(* Logix 5000 project; controller Wago_EtherNetIP_Adapter_Codesys35 vendor 1 type 14 code 196 rev 32.14; software revision 32.03 *)

TASK MainTask (continuous, watchdog 500 ms) : MainProgram

MODULES
   Local : vendor 1 type 14 code 196 (5069 0, rev 32.14)
      PFC200 : vendor 1285 type 12 code 120 (Ethernet 192.168.2.21, rev 1.1, StandardDataDriven RPI 20 ms)
END_MODULES

VAR_GLOBAL   (* controller tags *)
   AB_to_WAGO_DWORD : DINT := 100;   // DWORD DATA to WAGO PLC
   AB_to_WAGO_REAL : REAL := 7.2;   // REAL DATA to WAGO PLC
   WAGO_to_AB_DWORD : DINT := 500;   // DWORD Data From WAGO PLC
   WAGO_to_AB_REAL : REAL := 1000.0;   // REAL DATA from WAGO PLC
END_VAR

PROGRAM MainProgram   (* main routine MainRoutine *)

ROUTINE MainRoutine   (* ladder *)
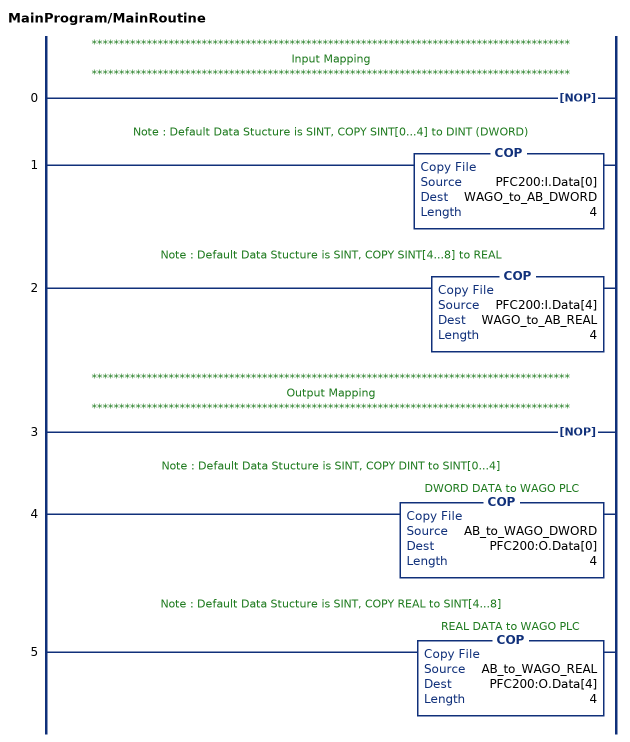
   // ***************************************************************************************
   // Input Mapping
   // ***************************************************************************************
   0: NOP();
   // Note : Default Data Stucture is SINT, COPY SINT[0...4] to DINT (DWORD)
   1: COP(PFC200:I.Data[0],WAGO_to_AB_DWORD,4);
   // Note : Default Data Stucture is SINT, COPY SINT[4...8] to REAL
   2: COP(PFC200:I.Data[4],WAGO_to_AB_REAL,4);
   // ***************************************************************************************
   // Output Mapping
   // ***************************************************************************************
   3: NOP();
   // Note : Default Data Stucture is SINT, COPY DINT to SINT[0...4]
   4: COP(AB_to_WAGO_DWORD,PFC200:O.Data[0],4);
   // Note : Default Data Stucture is SINT, COPY REAL to SINT[4...8]
   5: COP(AB_to_WAGO_REAL,PFC200:O.Data[4],4);
END_ROUTINE
END_PROGRAM
